(* PLC project Unnamed, Neznámo Unnamed 1 *)
(* stored: creationDateTime 2023-03-07T13:50:27, modificationDateTime 2023-03-07T14:34:24 *)

PROGRAM SFC_diagram
  VAR
    LocalVar0 : DINT;
  END_VAR

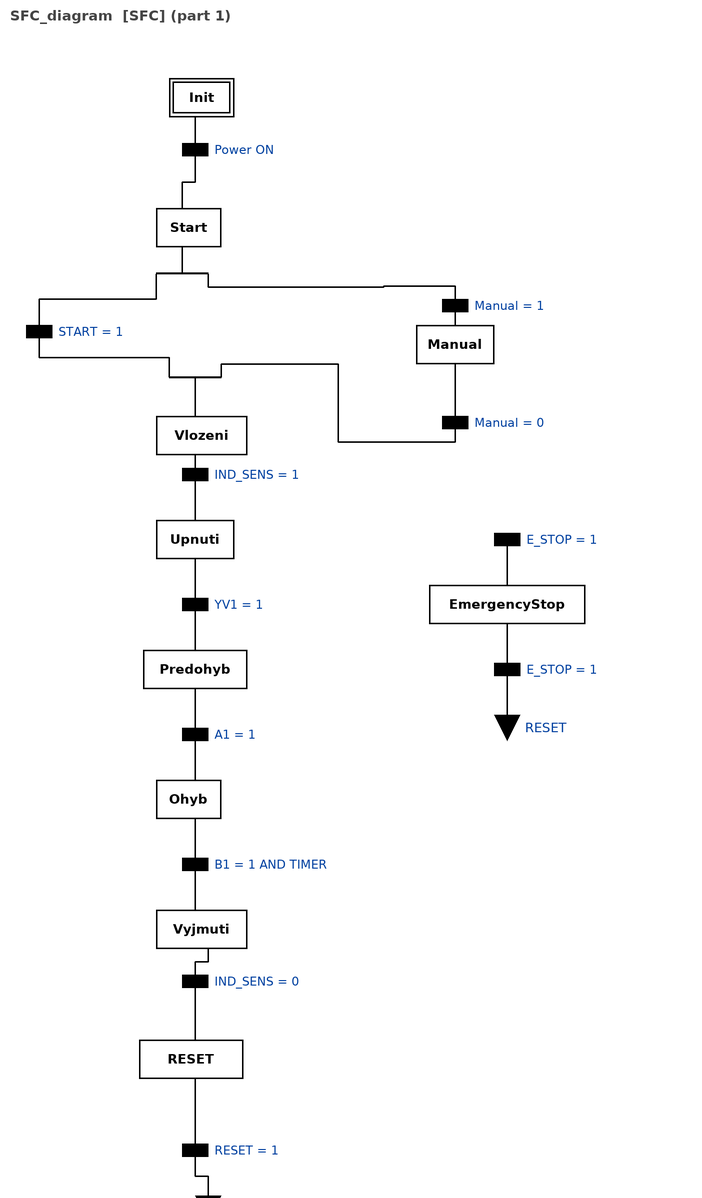
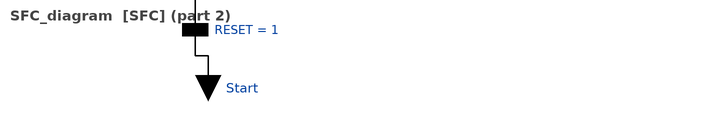
INITIAL_STEP Init:
END_STEP
TRANSITION FROM Init TO Start
  := Power ON;
END_TRANSITION
STEP Start:
END_STEP
TRANSITION FROM Start TO Vlozeni
  := START = 1;
END_TRANSITION
TRANSITION FROM Start TO Manual
  := Manual = 1;
END_TRANSITION
STEP Manual:
END_STEP
TRANSITION FROM Manual TO Vlozeni
  := Manual = 0;
END_TRANSITION
STEP Vlozeni:
END_STEP
TRANSITION FROM Vlozeni TO Upnuti
  := IND_SENS = 1;
END_TRANSITION
STEP Upnuti:
END_STEP
TRANSITION FROM Upnuti TO Predohyb
  := YV1 = 1;
END_TRANSITION
STEP EmergencyStop:
END_STEP
TRANSITION FROM EmergencyStop TO RESET
  := E_STOP = 1;
END_TRANSITION
STEP Predohyb:
END_STEP
TRANSITION FROM Predohyb TO Ohyb
  := A1 = 1;
END_TRANSITION
STEP Ohyb:
END_STEP
TRANSITION FROM Ohyb TO Vyjmuti
  := B1 = 1 AND TIMER;
END_TRANSITION
STEP Vyjmuti:
END_STEP
TRANSITION FROM Vyjmuti TO RESET
  := IND_SENS = 0;
END_TRANSITION
STEP RESET:
END_STEP
TRANSITION FROM RESET TO Start
  := RESET = 1;
END_TRANSITION
TRANSITION FROM ? TO EmergencyStop
  := E_STOP = 1;
END_TRANSITION
END_PROGRAM

CONFIGURATION Config0
  RESOURCE Res0 ON PLC
    TASK task0(INTERVAL := T#20ms, PRIORITY := 0);
    PROGRAM instance0 WITH task0 : SFC_diagram;
  END_RESOURCE
END_CONFIGURATION
